PROGRAM MAIN
VAR
	fbClk: FB_Clock;
END_VAR

fbClk(TIME_ON:= T#10MS, TIME_OFF:= T#200MS, OUT_CLK=> GVL.bClock);

END_PROGRAM

(* stored: Version 1.1.0.1, ProductVersion 3.1.4024.12
   POU MAIN: Id {b0810b71-a987-4dc5-8dba-9775a6550344}, SpecialFunc None *)
